FUNCTION_BLOCK FB_FrameFiforx
VAR_INPUT
	bLog		: BOOL := FALSE;
	stPut		: ST_FrameFifoEntrydatarx;
	
END_VAR
VAR_OUTPUT
	bOk			: BOOL;
	stGet		: ST_FrameFifoEntrydatarx;
	nCount		: UDINT := 0;
END_VAR
VAR
	fbBuffer 	: FB_MemRingBuffer;
	buffer		: ARRAY[0..NUMBER_OF_BYTE_FOR_ALL_FRAMEFIFO] OF BYTE;
	i : INT;
END_VAR
VAR CONSTANT
	SIZE_OF_FRAMEFIFO : UDINT := SIZEOF(ST_FrameFifoEntrydatarx);
	MAX_NUMBER_OF_FRAMEFIFO : UDINT := 10;
	NUMBER_OF_BYTE_FOR_ALL_FRAMEFIFO : UDINT := SIZE_OF_FRAMEFIFO*MAX_NUMBER_OF_FRAMEFIFO;
END_VAR

ACTION AddTail:
fbBuffer.A_AddTail( pBuffer:= ADR(buffer), cbBuffer:= SIZEOF(buffer),
					pWrite:= ADR( stPut ), cbWrite := SIZEOF( stPut ), 
					bOk=>bOk, nCount=>nCount );
END_ACTION

ACTION Clear:
FOR i:=0 TO RXDATASIZE BY 1 DO
stGet.rxdata[i] := 0;
END_FOR 

stGet.stRemoteAddr.nPort := 0;
stGet.stRemoteAddr.sAddr := '';
fbBuffer.A_Reset( pBuffer := ADR( buffer ), cbBuffer := SIZEOF( buffer ), 
					bOk=>bOk, nCount=>nCount );
END_ACTION

ACTION RemoveHead:
IF nCount = 0 THEN
	 
FOR i:=0 TO RXDATASIZE BY 1 DO
stGet.rxdata[i] := 0;
END_FOR 

	stGet.stRemoteAddr.nPort := 0;
	stGet.stRemoteAddr.sAddr := '';
	bOk := FALSE;
	RETURN;
END_IF

fbBuffer.A_RemoveHead( pBuffer:= ADR(buffer), cbBuffer:= SIZEOF(buffer),
						pRead := ADR( stGet ), cbRead := SIZEOF( stGet ),
						bOk=>bOk, nCount=>nCount );
END_ACTION

END_FUNCTION_BLOCK

(* stored: Version 1.1.0.1, ProductVersion 3.1.4024.13
   POU FB_FrameFiforx: Id {becbd2a1-a819-4aec-890c-7789c9c38fdd}, SpecialFunc None
   Action AddTail: Id {8cdf03d3-64b2-45ae-a264-11610aad1642}
   Action Clear: Id {26ab6ca5-646d-425c-83d1-b0188477fda2}
   Action RemoveHead: Id {96e97635-d9c5-4b62-8973-13186b34b7ff} *)
